// TIA Portal V17 export
// export: Created 2022-03-12T16:05:35.1222026Z, ExportSetting WithDefaults, DisplayName Totally Integrated Automation Portal, DisplayVersion V17, DisplayName TIA Portal Openness, DisplayVersion V17, DisplayName TIA Portal Version Control Interface, DisplayVersion V17, DisplayName STEP 7 Professional, DisplayVersion V17, DisplayName STEP 7 Safety, DisplayVersion V17, DisplayName WinCC Advanced / Unified PC, DisplayVersion V17
TYPE "typeLPMLV30_Configuration"
TITLE = typeLPMLV30_Configuration
// Support: tech.team.motioncontrol@siemens.com 
// Fax: +49 (0) 9131/98-1297
// stored: IsFailsafeCompliant false
   STRUCT
      disabledUnitModes : Array[0.."LPMLV30_MAX_MODES_UPPER_LIM"] of Bool;   // TRUE: Disable unit mode xx
      disabledStatesInUnitModes : Array[0.."LPMLV30_MAX_MODES_UPPER_LIM"] of DInt;   // TRUE: Disable states in unit mode (bit number = state number)
   END_STRUCT;
   // disabledUnitModes[0..11] := false;
   // disabledUnitModes[12..31] := true;
   // disabledStatesInUnitModes[0..31] := 0;
END_TYPE
